{attribute 'qualified_only'}
VAR_GLOBAL
	
fRealValue : REAL;

END_VAR

(* stored: Version 1.1.0.1, ProductVersion 3.1.4024.12
   GVL GVL: Id {61ebd7ca-2d10-4572-b60b-7596713c407d} *)
